// TIA Portal V20 export
DATA_BLOCK "InstCallGlobal"   // DB265
// stored: InstanceOfName CallGlobal, InstanceOfType FB
"CallGlobal"
   // VAR
   //    statClockSysMemOld { ExternalWritable := 'False'} : Byte;
   //    statRev0Hz5 : Bool;
   //    statTonTimer : Array[0..1] of IEC_TIMER;
   //    instLAF_PowerOnOff { ExternalWritable := 'False'} : "LAF_PowerOnOff";
   //    instLAF_HmiHeaderManager { ExternalWritable := 'False'} : "LAF_HmiHeaderManager";
   //    instLAF_ClockGen { ExternalWritable := 'False'} : "LAF_ClockGenerator";
   //    instLSNTP_Server { ExternalWritable := 'False'} : "LSNTP_Server";
   //    instRemoteAccess { ExternalWritable := 'False'} : "LRemoteAccess_MobilePanelMonitor";
   //    statPulse : Array[0..99] of Bool;
   // END_VAR
BEGIN
   instLSNTP_Server.statConParam.InterfaceId := 72;
END_DATA_BLOCK
